FUNCTION_BLOCK FB_RFID
VAR_INPUT
	cmd					: E_RFIDCommand := E_RFIDCommand.None;
	cmdReset			: BOOL;
	inpSimID			: STRING := '12345';
	
	inpSim				: BOOL := TRUE;
	inpID				AT %I* : STRING;
END_VAR
VAR_OUTPUT
	stsState			: E_RFIDState := E_RFIDState.Idle;
	stsFaultCode		: DINT;
	stsCurrentID		: STRING;
	
	outScan				AT %Q* : BOOL;
	outResetScanner		AT %Q* : BOOL;
END_VAR
VAR
	ReadTimer			: TON;
	ReadSimTime			: TIME := T#5S;
	ReadFailTime		: TIME := T#30S;
END_VAR
VAR CONSTANT
	NULL_ID				: STRING := '';
END_VAR

Faults();
StateMachine();
Control();

METHOD Control : BOOL
VAR_INPUT
END_VAR
outScan := stsState = E_RFIDState.Reading;
outResetScanner := stsState = E_RFIDState.Completing;
END_METHOD

METHOD Faults : BOOL
VAR_INPUT
END_VAR
ReadTimer(IN := stsState = E_RFIDState.Reading, PT := ReadFailTime);
IF ReadTimer.Q THEN
	stsFaultCode := 100;
ELSE
	stsFaultCode := 0;
END_IF
END_METHOD

METHOD Simulate : BOOL
VAR_INPUT
END_VAR
IF outScan AND ReadTimer.ET >= ReadSimTime THEN
	inpID := inpSimID;
END_IF

IF outResetScanner THEN
	inpID := NULL_ID;
END_IF
END_METHOD

METHOD StateMachine : BOOL
VAR_INPUT
END_VAR
IF inpSim THEN
	Simulate();
END_IF

CASE stsState OF
	E_RFIDState.Idle:
		IF cmd = E_RFIDCommand.Clear THEN
			stsState := E_RFIDState.Clearing;
		ELSIF cmd = E_RFIDCommand.Read THEN
			stsState := E_RFIDState.Reading;
		END_IF
	E_RFIDState.Clearing:
		stsCurrentID := NULL_ID;
		IF stsCurrentID = NULL_ID THEN
			stsState := E_RFIDState.Idle;
		END_IF
	E_RFIDState.Reading:
		IF inpID <> NULL_ID THEN
			stsCurrentID := inpID;
			stsState := E_RFIDState.Completing;
		ELSIF stsFaultCode <> 0 AND cmdReset THEN
			stsState := E_RFIDState.Idle;
		END_IF
	E_RFIDState.Completing:
		IF inpID = NULL_ID THEN
			stsState := E_RFIDState.Idle;
		END_IF
END_CASE

cmd := E_RFIDCommand.None;
cmdReset := FALSE;
END_METHOD

END_FUNCTION_BLOCK

(* stored: Version 1.1.0.1, ProductVersion 3.1.4024.4
   POU FB_RFID: Id {e37777d5-682f-4821-a127-0aa1343bd3d1}, SpecialFunc None
   Method Control: Id {e99bc787-ec25-45fe-8ec4-b88288f601a9}
   Method Faults: Id {5fb03235-7ce4-4e94-b30b-b11285540766}
   Method Simulate: Id {e29c3a32-e4a7-4a46-ac28-92030b00d33a}
   Method StateMachine: Id {ed3a31f4-422a-4189-9a24-e0b9748aaeb1} *)
